TYPE DOutputs :
STRUCT
	output1 : BOOL;
	output2 : BOOL;
	output3 : BOOL;
	output4 : BOOL;
	controlOutput1 : BOOL;
	controlOutput2 : BOOL;
	controlOutput3 : BOOL;
	controlOutput4 : BOOL;
END_STRUCT
END_TYPE

(* stored: Version 1.1.0.1, ProductVersion 3.1.4024.9
   DUT DOutputs: Id {fbcbb2f6-384f-441c-9553-bfbd32af245f} *)
